LIN {X 0,Y 54.915,Z 334.907,A -85,B 0,C 180,E1 -31667.388,E2 -31667.388} C_VEL
LIN {X 0,Y 62.069,Z 323.757,A -85,B 0,C 180,E1 -31667.589,E2 -31667.589} C_VEL
LIN {X 0,Y 65.376,Z 317.558,A -85,B 0,C 180,E1 -31667.617,E2 -31667.617} C_VEL
LIN {X 0,Y 69.157,Z 318.45,A -85,B 0,C 180,E1 -31667.838,E2 -31667.838} C_VEL
LIN {X 0,Y 69.157,Z 600,A -85,B 0,C 180,E1 -31667.838,E2 -31667.838} C_VEL
LIN {X 0,Y 69.157,Z 600,A -85,B 0,C 180,E1 -31667.838,E2 -31667.838}

QRS_NEXT_CUT()

QRS_NEXT()
QRS_HOME()

END
